FUNCTION_BLOCK SocketCloseTask
VAR_INPUT
END_VAR
VAR_OUTPUT
END_VAR
VAR
END_VAR

END_FUNCTION_BLOCK

(* stored: Version 1.1.0.1, ProductVersion 3.1.4024.12
   POU SocketCloseTask: Id {a9ec101e-14e7-48c3-bce3-b5c9494e4a85}, SpecialFunc None *)
